KUKA KRL program: var_proxy_v2.src, var_proxy_v2.dat

--- var_proxy_v2.src ---
&ACCESS RVP
&REL 159
&PARAM EDITMASK = *
&PARAM TEMPLATE = C:\KRC\Roboter\Template\ExpertVorgabe
DEF var_proxy_v2( )
ghCommand.motiontype = 0
ghCommand.speed = 10

WAIT SEC 1.0 ;

;FOLD INI

  ;FOLD BASISTECH INI
    GLOBAL INTERRUPT DECL 3 WHEN $STOPMESS==TRUE DO IR_STOPM ( )
    INTERRUPT ON 3
    BAS (#INITMOV,0 )
  ;ENDFOLD (BASISTECH INI)
  ;FOLD USER INI
    ;Make your modifications here

  ;ENDFOLD (USER INI)
;ENDFOLD (INI)


LOOP


$ADVANCE =1;

SWITCH ghCommand.motionType
    CASE 1
        msgnotify("motion type 1 - jnt ")
       ;DO NOT USE "CHANGE" on tp for the next line; See the detail under open fold
;FOLD PTP jntPos Vel=100 % PDAT3 Tool[1]:DFM24_SPIKE Base[1]:DFM24_BASE;%{PE}%R 8.3.38,%MKUKATPBASIS,%CMOVE,%VPTP,%P 1:PTP, 2:jntPos, 3:, 5:100, 7:PDAT3
$BWDSTART=FALSE
PDAT_ACT=PPDAT3
FDAT_ACT=FjntPos
BAS(#PTP_PARAMS,ghCommand.speed)
PTP ghCommand.jntPos
;ENDFOLD
      ghCommand.motionType = 0

    CASE 2
        msgnotify("motion type 2 - linear ")
        PTP $AXIS_ACT
        ghMotionBuf = ghCommand.targetPos
        IF (VARSTATE("ghCommand.targetPos.S")<>#INITIALIZED) THEN
           ghMotionBuf.S = $POS_ACT.S
           ghMotionBuf.T = $POS_ACT.T

        ENDIF
        ; DO NOT USE "CHANGE" on tp for the next line; See the detail under open fold
;FOLD LIN p7 Vel=2 m/s CPDAT2 Tool[1]:DFM24_SPIKE Base[1]:DFM24_BASE;%{PE}%R 8.3.38,%MKUKATPBASIS,%CMOVE,%VLIN,%P 1:LIN, 2:p7, 3:, 5:2, 7:CPDAT2
$BWDSTART=FALSE
LDAT_ACT=LCPDAT2
FDAT_ACT=Fp7
BAS(#CP_PARAMS,ghCommand.speed)
LIN ghMotionBuf

;ENDFOLD
       ghCommand.motionType = 0
    CASE 3
         msgnotify("cmd type 3 - setting do")
         $OUT[ghCommand.do_address] = ghCommand.do_value
         ghCommand.motionType=0
    DEFAULT
        msgnotify("waiting next cmd");
        WAIT SEC 1.0;
ENDSWITCH
ENDLOOP

END

--- var_proxy_v2.dat ---
&ACCESS RVP
&REL 159
&PARAM EDITMASK = *
&PARAM TEMPLATE = C:\KRC\Roboter\Template\ExpertVorgabe
DEFDAT  var_proxy_v2 PUBLIC
GLOBAL STRUC MotionCommand INT motionType,E6AXIS jntPos,E6POS targetPos,REAL speed, INT do_address, BOOL do_value

DECL MotionCommand ghCommand
DECL E6POS ghMotionBuf






DECL BASIS_SUGG_T LAST_BASIS={POINT1[] "jntPos                  ",POINT2[] "jntPos                  ",CP_PARAMS[] "CPDAT2                  ",PTP_PARAMS[] "PDAT4                   ",CONT[] "                        ",CP_VEL[] "2                       ",PTP_VEL[] "100                     ",SYNC_PARAMS[] "SYNCDAT                 ",SPL_NAME[] "S0                      ",A_PARAMS[] "ADAT0                   "}
DECL FDAT FP1={TOOL_NO 1,BASE_NO 1,IPO_FRAME #BASE,POINT2[] " ",TQ_STATE FALSE}
DECL PDAT PPDAT1={VEL 100.000,ACC 100.000,APO_DIST 100.000,GEAR_JERK 50.0000,EXAX_IGN 0}
DECL E6POS XP2={X 764.445740,Y -1158.58606,Z 1531.21252,A -63.2373352,B -7.46904755,C -80.2913895,S 22,T 19,E1 3127.46094,E2 0.0,E3 0.0,E4 0.0,E5 0.0,E6 0.0}
DECL FDAT FP2={TOOL_NO 1,BASE_NO 1,IPO_FRAME #BASE,POINT2[] " ",TQ_STATE FALSE}
DECL PDAT PPDAT2={VEL 100.000,ACC 100.000,APO_DIST 100.000,GEAR_JERK 50.0000,EXAX_IGN 0}
DECL E6POS XP3={X 764.445740,Y -1158.58606,Z 1531.21252,A -63.2373352,B -7.46904755,C -80.2913895,S 22,T 19,E1 3127.46094,E2 0.0,E3 0.0,E4 0.0,E5 0.0,E6 0.0}
DECL FDAT FP3={TOOL_NO 1,BASE_NO 1,IPO_FRAME #BASE,POINT2[] " ",TQ_STATE FALSE}
DECL LDAT LCPDAT1={VEL 2.00000,ACC 100.000,APO_DIST 100.000,APO_FAC 50.0000,AXIS_VEL 100.000,AXIS_ACC 100.000,ORI_TYP #VAR,CIRC_TYP #BASE,JERK_FAC 50.0000,GEAR_JERK 50.0000,EXAX_IGN 0}
DECL E6POS XP4={X 811.273315,Y -1374.55237,Z 1651.36218,A -63.9521332,B -6.23386812,C -82.2733307,S 22,T 19,E1 2821.00,E2 0.0,E3 0.0,E4 0.0,E5 0.0,E6 0.0}
DECL E6POS XP6={X 104.214714,Y -1710.04883,Z 1411.98376,A -179.136917,B -0.170715928,C 179.671097,S 18,T 42,E1 3200.00,E2 0.0,E3 0.0,E4 0.0,E5 0.0,E6 0.0}
DECL FDAT Fp6={TOOL_NO 1,BASE_NO 1,IPO_FRAME #BASE,POINT2[] " ",TQ_STATE FALSE}
DECL LDAT LCPDAT2={VEL 2.00000,ACC 100.000,APO_DIST 100.000,APO_FAC 50.0000,AXIS_VEL 100.000,AXIS_ACC 100.000,ORI_TYP #VAR,CIRC_TYP #BASE,JERK_FAC 50.0000,GEAR_JERK 50.0000,EXAX_IGN 0}
DECL E6POS XP7={X 104.214714,Y -1710.04883,Z 1411.98376,A -179.136917,B -0.170715928,C 179.671097,S 18,T 2,E1 3200.00,E2 0.0,E3 0.0,E4 0.0,E5 0.0,E6 0.0}
DECL FDAT Fp7={TOOL_NO 1,BASE_NO 1,IPO_FRAME #BASE,POINT2[] " ",TQ_STATE FALSE}
DECL PDAT PPDAT3={VEL 100.000,ACC 100.000,APO_DIST 100.000,GEAR_JERK 50.0000,EXAX_IGN 0}
DECL E6POS XJNTPOS={X 104.214714,Y -1710.04883,Z 1411.98376,A -179.136917,B -0.170715928,C 179.671097,S 18,T 42,E1 3200.00,E2 0.0,E3 0.0,E4 0.0,E5 0.0,E6 0.0}
DECL FDAT FjntPos={TOOL_NO 1,BASE_NO 1,IPO_FRAME #BASE,POINT2[] " ",TQ_STATE FALSE}
DECL PDAT PPDAT4={VEL 100.000,ACC 100.000,APO_DIST 100.000,GEAR_JERK 50.0000,EXAX_IGN 0}
ENDDAT
